TYPE OUTPUT :
STRUCT
END_STRUCT
END_TYPE

(* stored: Version 1.1.0.1, ProductVersion 3.1.4024.4
   DUT OUTPUT: Id {79f743cb-b0c8-4ef7-b469-ce78aee8168e} *)
